// TIA Portal V16 export
// export: Created 2021-09-08T12:46:11.6644631Z, ExportSetting WithDefaults, DisplayName Totally Integrated Automation Portal, DisplayVersion V16 Update 3, DisplayName TIA Portal Version Control Interface, DisplayVersion V16 Update 2, DisplayName TIA Portal Openness, DisplayVersion V16 Update 3, DisplayName TIA Portal Teamcenter Gateway, DisplayVersion V16, DisplayName STEP 7 Professional, DisplayVersion V16 Update 3, DisplayName STEP 7 Safety, DisplayVersion V16, DisplayName WinCC Advanced, DisplayVersion V16 Update 3
FUNCTION_BLOCK "AllPump"   // FB2, FBD
{ S7_Optimized_Access := 'TRUE' }
VERSION : 0.1
// stored: AutoNumber true, IsIECCheckEnabled false, IsRetainMemResEnabled false, MemoryReserve 100, SetENOAutomatically false, UDAEnableTagReadback false
   VAR
      PU30x { S7_SetPoint := 'True'} : "PumpCntrl2Pu1Fc";
      cmUZ_P30x { S7_SetPoint := 'True'} : Bool;
      cmUZ_P120x : Bool;
      cmUZ_P150x : Bool;
      tmrLowPresP30x { S7_SetPoint := 'True'} : TON_TIME;
      tmrLowFreqP30x { S7_SetPoint := 'True'} : TON_TIME;
      tLowPresP30x { S7_SetPoint := 'True'} : Time;
      tLowFreqP30x : Time;
      PU120x { S7_SetPoint := 'True'} : "PumpCntrl2Pu1Fc";
      tmrLowPresP120x { S7_SetPoint := 'True'} : TON_TIME;
      tLowPresP120x { S7_SetPoint := 'True'} : Time;
      tNoPulseP120x : Time;
      PU150x { S7_SetPoint := 'True'} : "PumpCntrl2Pu1Fc";
      tmrLowPresP150x { S7_SetPoint := 'True'} : TON_TIME;
      tLowPresP150x { S7_SetPoint := 'True'} : Time;
      tNoPulseP150x : Time;
      noPulseTOF_P120x { S7_SetPoint := 'True'} : "noPulseTOF";
      noPulseTOF_P150x { S7_SetPoint := 'True'} : "noPulseTOF";
      P701 { S7_SetPoint := 'True'} : "PumpCntr";
      P702 { S7_SetPoint := 'True'} : "PumpCntr";
      P901 { S7_SetPoint := 'True'} : "PumpCntr";
      P1301 { S7_SetPoint := 'True'} : "PumpCntr";
      P2001 { S7_SetPoint := 'True'} : "PumpCntr";
      C501 { S7_SetPoint := 'True'} : "PumpCntr";
      sel2pu_P70x { S7_SetPoint := 'True'} : "sel2pu";
   END_VAR
BEGIN

REGION Network 1: P30x - выбор рабочего
   // Помилка датчиків рівня TW201, TW202
   // Аварійно низький рівень TW201, TW202
   // Помилка датчика PT301
   // Аварійно низьке значення PT301
   // Аварійно високе значення PT301
   // Помилка датчика PT401
   // Аварійно низьке значення PT401
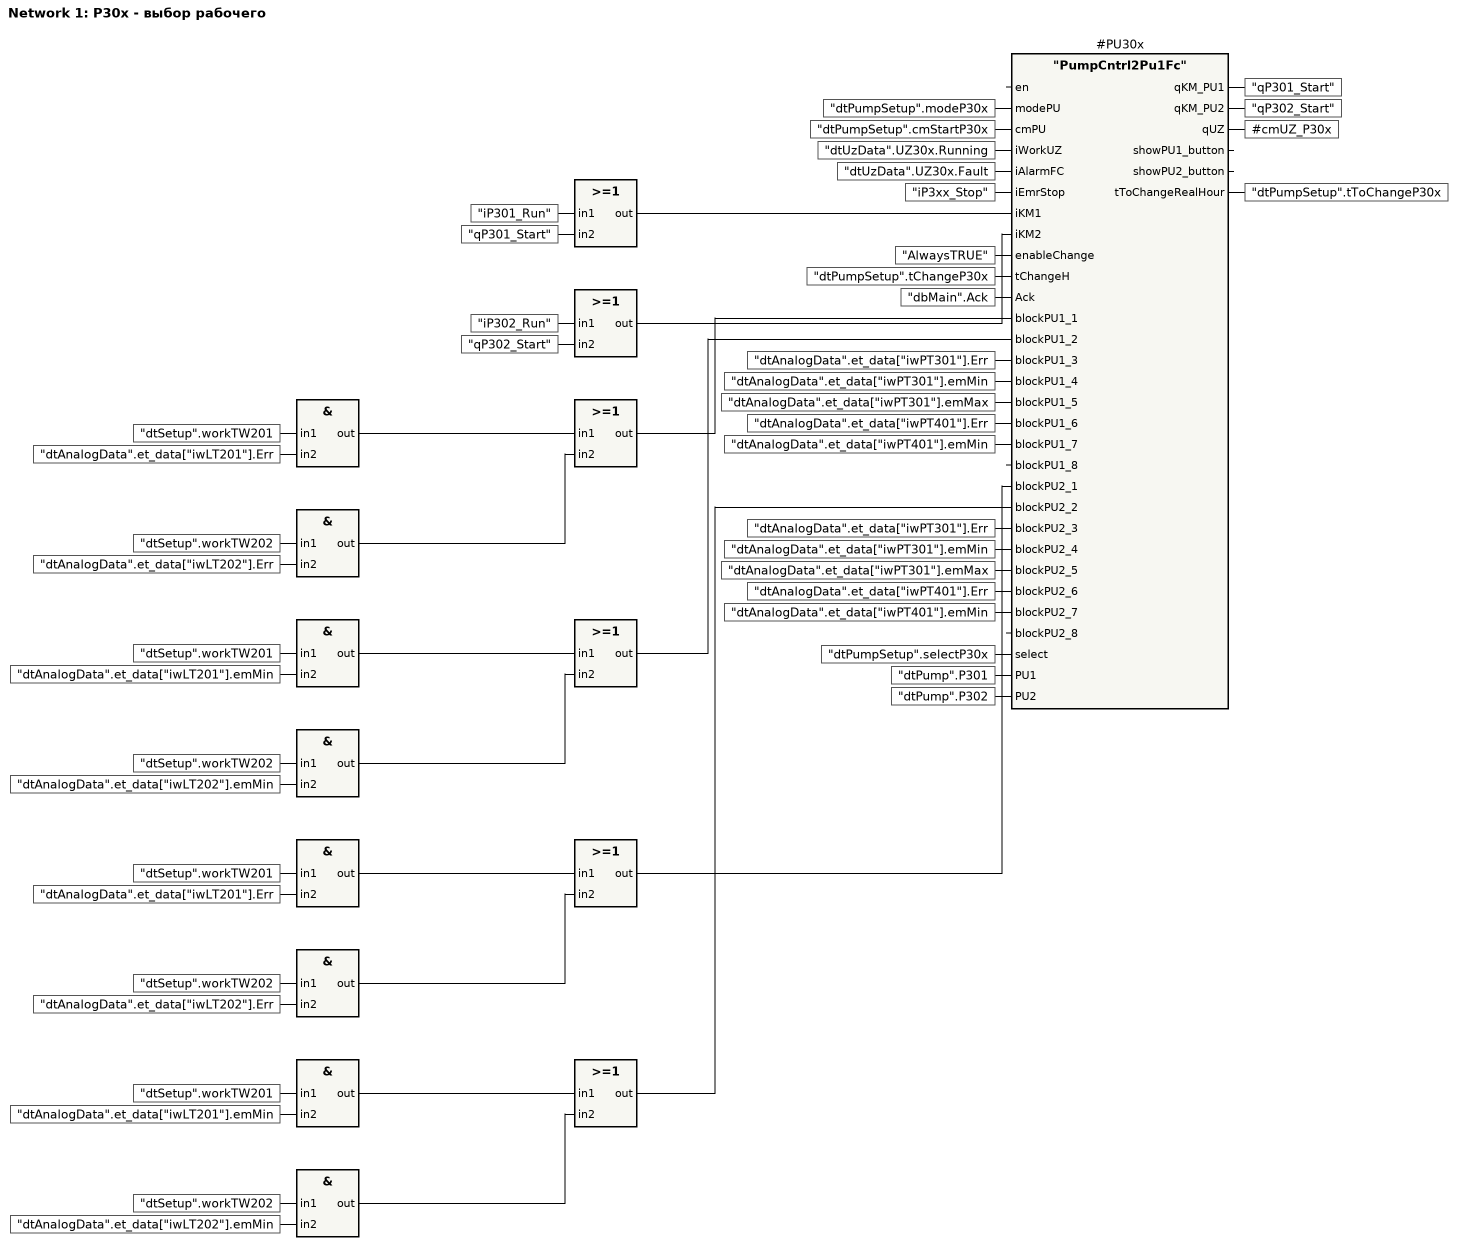
   #PU30x(modePU := "dtPumpSetup".modeP30x,   // "PumpCntrl2Pu1Fc"
          cmPU := "dtPumpSetup".cmStartP30x,
          iWorkUZ := "dtUzData".UZ30x.Running,
          iAlarmFC := "dtUzData".UZ30x.Fault,
          iEmrStop := "iP3xx_Stop",
          iKM1 := "iP301_Run" OR "qP301_Start",
          iKM2 := "iP302_Run" OR "qP302_Start",
          enableChange := "AlwaysTRUE",
          tChangeH := "dtPumpSetup".tChangeP30x,
          Ack := "dbMain".Ack,
          blockPU1_1 := ("dtSetup".workTW201 AND "dtAnalogData".et_data["iwLT201"].Err) OR ("dtSetup".workTW202 AND "dtAnalogData".et_data["iwLT202"].Err),
          blockPU1_2 := ("dtSetup".workTW201 AND "dtAnalogData".et_data["iwLT201"].emMin) OR ("dtSetup".workTW202 AND "dtAnalogData".et_data["iwLT202"].emMin),
          blockPU1_3 := "dtAnalogData".et_data["iwPT301"].Err,
          blockPU1_4 := "dtAnalogData".et_data["iwPT301"].emMin,
          blockPU1_5 := "dtAnalogData".et_data["iwPT301"].emMax,
          blockPU1_6 := "dtAnalogData".et_data["iwPT401"].Err,
          blockPU1_7 := "dtAnalogData".et_data["iwPT401"].emMin,
          blockPU2_1 := ("dtSetup".workTW201 AND "dtAnalogData".et_data["iwLT201"].Err) OR ("dtSetup".workTW202 AND "dtAnalogData".et_data["iwLT202"].Err),
          blockPU2_2 := ("dtSetup".workTW201 AND "dtAnalogData".et_data["iwLT201"].emMin) OR ("dtSetup".workTW202 AND "dtAnalogData".et_data["iwLT202"].emMin),
          blockPU2_3 := "dtAnalogData".et_data["iwPT301"].Err,
          blockPU2_4 := "dtAnalogData".et_data["iwPT301"].emMin,
          blockPU2_5 := "dtAnalogData".et_data["iwPT301"].emMax,
          blockPU2_6 := "dtAnalogData".et_data["iwPT401"].Err,
          blockPU2_7 := "dtAnalogData".et_data["iwPT401"].emMin,
          select := "dtPumpSetup".selectP30x,
          PU1 := "dtPump".P301,
          PU2 := "dtPump".P302,
          qKM_PU1 => "qP301_Start",
          qKM_PU2 => "qP302_Start",
          qUZ => #cmUZ_P30x,
          tToChangeRealHour => "dtPumpSetup".tToChangeP30x);
END_REGION

REGION Network 2: P30x - частотник
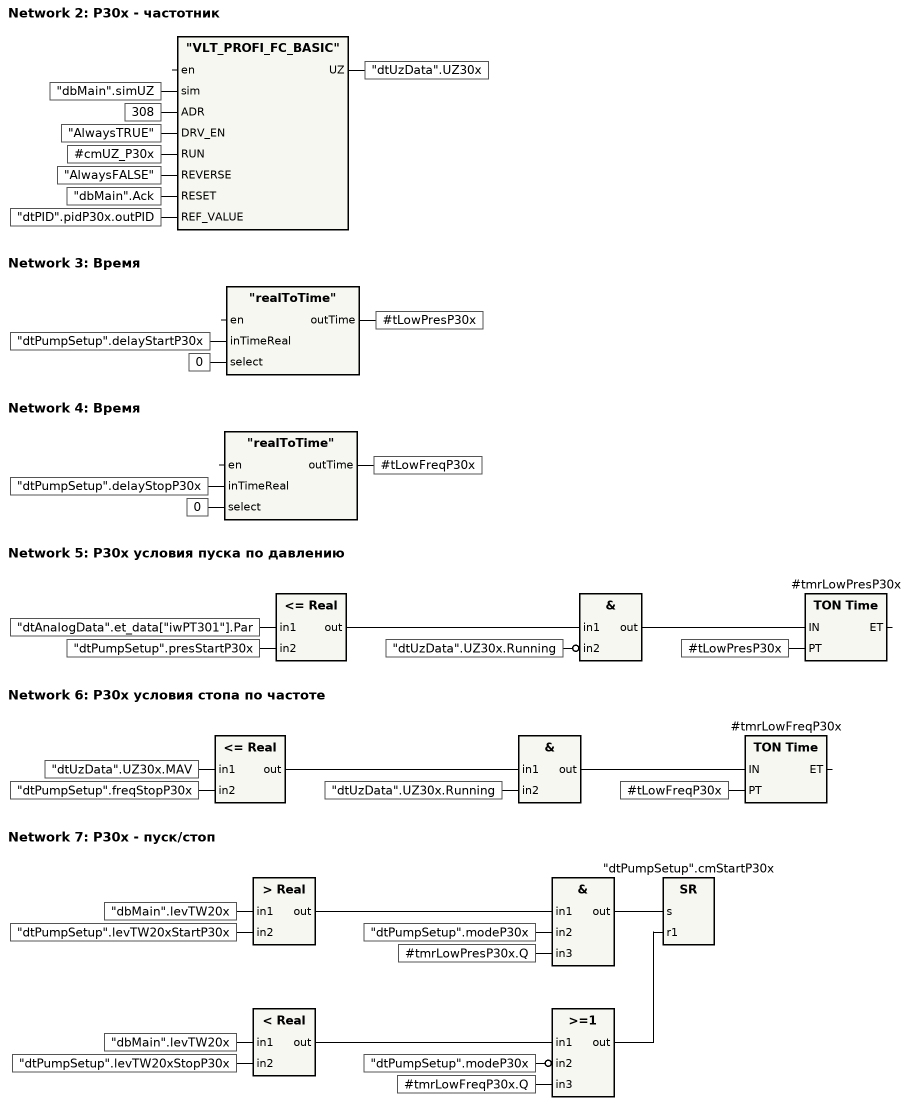
   "VLT_PROFI_FC_BASIC"(sim := "dbMain".simUZ,
                        ADR := 308,
                        DRV_EN := "AlwaysTRUE",
                        RUN := #cmUZ_P30x,
                        REVERSE := "AlwaysFALSE",
                        RESET := "dbMain".Ack,
                        REF_VALUE := "dtPID".pidP30x.outPID,
                        UZ => "dtUzData".UZ30x);
END_REGION

REGION Network 3: Время
   "realToTime"(inTimeReal := "dtPumpSetup".delayStartP30x, select := 0, outTime => #tLowPresP30x);
END_REGION

REGION Network 4: Время
   "realToTime"(inTimeReal := "dtPumpSetup".delayStopP30x, select := 0, outTime => #tLowFreqP30x);
END_REGION

REGION Network 5: P30x условия пуска по давлению
   #tmrLowPresP30x(IN := ("dtAnalogData".et_data["iwPT301"].Par <= "dtPumpSetup".presStartP30x) AND NOT "dtUzData".UZ30x.Running,   // TON
                   PT := #tLowPresP30x);
END_REGION

REGION Network 6: P30x условия стопа по частоте
   #tmrLowFreqP30x(IN := ("dtUzData".UZ30x.MAV <= "dtPumpSetup".freqStopP30x) AND "dtUzData".UZ30x.Running,   // TON
                   PT := #tLowFreqP30x);
END_REGION

REGION Network 7: P30x - пуск/стоп
   IF ("dbMain".levTW20x > "dtPumpSetup".levTW20xStartP30x) AND "dtPumpSetup".modeP30x AND #tmrLowPresP30x.Q THEN
       "dtPumpSetup".cmStartP30x := TRUE;   // SR flip-flop
   END_IF;
   IF ("dbMain".levTW20x < "dtPumpSetup".levTW20xStopP30x) OR NOT "dtPumpSetup".modeP30x OR #tmrLowFreqP30x.Q THEN
       "dtPumpSetup".cmStartP30x := FALSE;
   END_IF;
END_REGION

REGION Network 8: -------------------------------------------------P1201, 1202
END_REGION

REGION Network 9: P120x - выбор рабочего !!!!!!!!!!!!!!!!!!!!!!!!!!!!!!!!!!!!!!!!!!!!!!!!!! Убрать iP1201_run
   // Помилка датчиків рівня LT1101
   // Аварійно низький рівень TW1101
   // Помилка датчика PT1201
   // Аварійно низьке значення PT1201
   // Аварійно високе значення PT1201
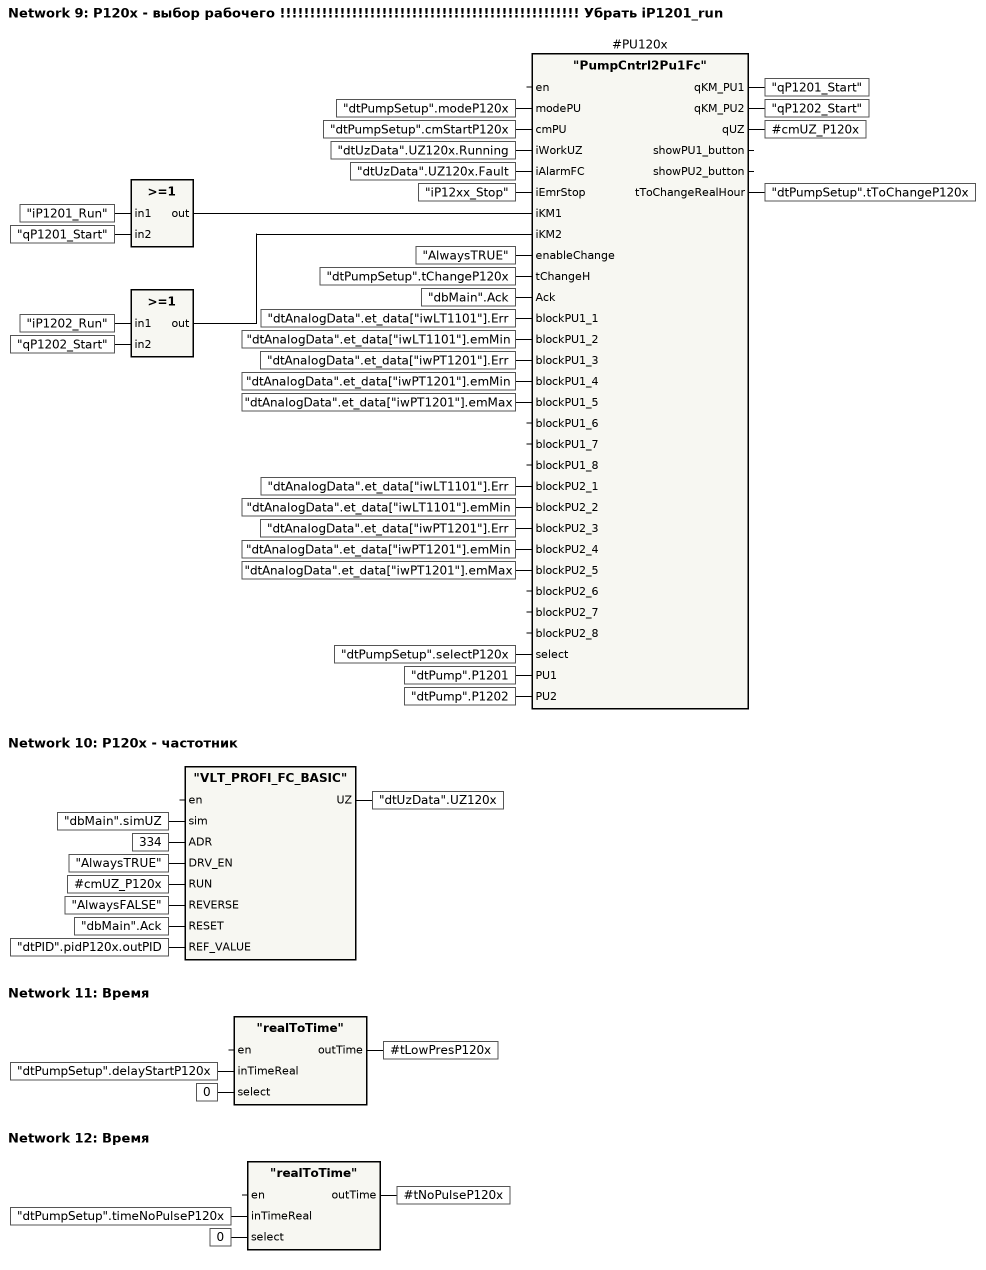
   #PU120x(modePU := "dtPumpSetup".modeP120x,   // "PumpCntrl2Pu1Fc"
           cmPU := "dtPumpSetup".cmStartP120x,
           iWorkUZ := "dtUzData".UZ120x.Running,
           iAlarmFC := "dtUzData".UZ120x.Fault,
           iEmrStop := "iP12xx_Stop",
           iKM1 := "iP1201_Run" OR "qP1201_Start",
           iKM2 := "iP1202_Run" OR "qP1202_Start",
           enableChange := "AlwaysTRUE",
           tChangeH := "dtPumpSetup".tChangeP120x,
           Ack := "dbMain".Ack,
           blockPU1_1 := "dtAnalogData".et_data["iwLT1101"].Err,
           blockPU1_2 := "dtAnalogData".et_data["iwLT1101"].emMin,
           blockPU1_3 := "dtAnalogData".et_data["iwPT1201"].Err,
           blockPU1_4 := "dtAnalogData".et_data["iwPT1201"].emMin,
           blockPU1_5 := "dtAnalogData".et_data["iwPT1201"].emMax,
           blockPU2_1 := "dtAnalogData".et_data["iwLT1101"].Err,
           blockPU2_2 := "dtAnalogData".et_data["iwLT1101"].emMin,
           blockPU2_3 := "dtAnalogData".et_data["iwPT1201"].Err,
           blockPU2_4 := "dtAnalogData".et_data["iwPT1201"].emMin,
           blockPU2_5 := "dtAnalogData".et_data["iwPT1201"].emMax,
           select := "dtPumpSetup".selectP120x,
           PU1 := "dtPump".P1201,
           PU2 := "dtPump".P1202,
           qKM_PU1 => "qP1201_Start",
           qKM_PU2 => "qP1202_Start",
           qUZ => #cmUZ_P120x,
           tToChangeRealHour => "dtPumpSetup".tToChangeP120x);
END_REGION

REGION Network 10: P120x - частотник
   "VLT_PROFI_FC_BASIC"(sim := "dbMain".simUZ,
                        ADR := 334,
                        DRV_EN := "AlwaysTRUE",
                        RUN := #cmUZ_P120x,
                        REVERSE := "AlwaysFALSE",
                        RESET := "dbMain".Ack,
                        REF_VALUE := "dtPID".pidP120x.outPID,
                        UZ => "dtUzData".UZ120x);
END_REGION

REGION Network 11: Время
   "realToTime"(inTimeReal := "dtPumpSetup".delayStartP120x, select := 0, outTime => #tLowPresP120x);
END_REGION

REGION Network 12: Время
   "realToTime"(inTimeReal := "dtPumpSetup".timeNoPulseP120x, select := 0, outTime => #tNoPulseP120x);
END_REGION

REGION Network 13: P120x условия пуска по давлению
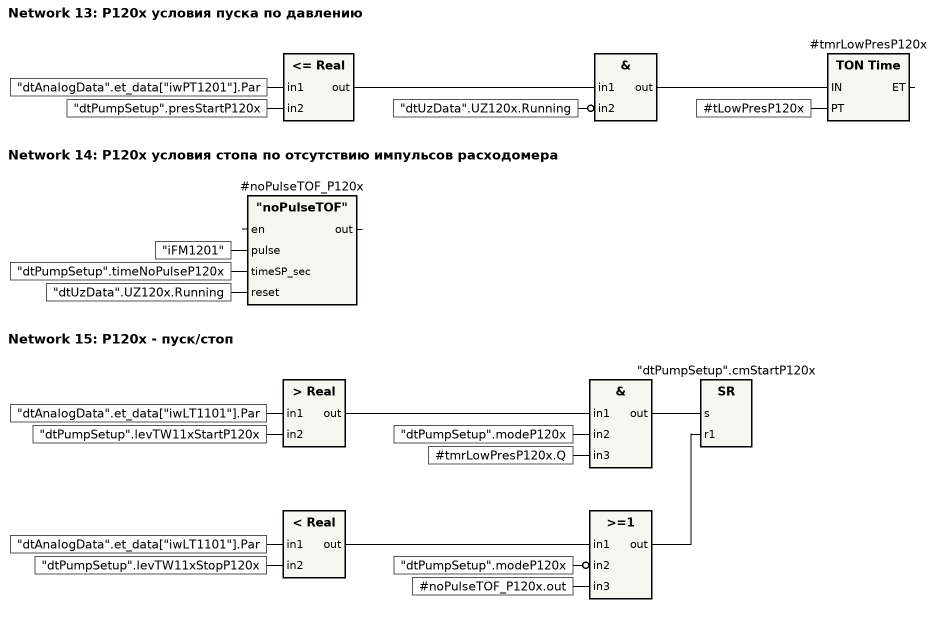
   #tmrLowPresP120x(IN := ("dtAnalogData".et_data["iwPT1201"].Par <= "dtPumpSetup".presStartP120x) AND NOT "dtUzData".UZ120x.Running,   // TON
                    PT := #tLowPresP120x);
END_REGION

REGION Network 14: P120x условия стопа по отсутствию импульсов расходомера
   #noPulseTOF_P120x(pulse := "iFM1201",   // "noPulseTOF"
                     timeSP_sec := "dtPumpSetup".timeNoPulseP120x,
                     reset := "dtUzData".UZ120x.Running);
END_REGION

REGION Network 15: P120x - пуск/стоп
   IF ("dtAnalogData".et_data["iwLT1101"].Par > "dtPumpSetup".levTW11xStartP120x) AND "dtPumpSetup".modeP120x AND #tmrLowPresP120x.Q THEN
       "dtPumpSetup".cmStartP120x := TRUE;   // SR flip-flop
   END_IF;
   IF ("dtAnalogData".et_data["iwLT1101"].Par < "dtPumpSetup".levTW11xStopP120x) OR NOT "dtPumpSetup".modeP120x OR #noPulseTOF_P120x.out THEN
       "dtPumpSetup".cmStartP120x := FALSE;
   END_IF;
END_REGION

REGION Network 16: -------------------------------------------------P1501, 1502
END_REGION

REGION Network 17: P150x - выбор рабочего !!!!!!!!!!!!!!!!!!!!!!!!!!!!!!!!!!!!!!!!!!!!!!!!!! Убрать iP1501_run
   // Помилка датчиків рівня TW1401, TW1402
   // Аварійно низький рівень TW1401, TW1402
   // Помилка датчика PT1501
   // Аварійно низьке значення PT1501
   // Аварійно високе значення PT1501
   // Помилка датчика PT1701
   // Аварійно низьке значення PT1701
   // Аварійно високе значення PT1701
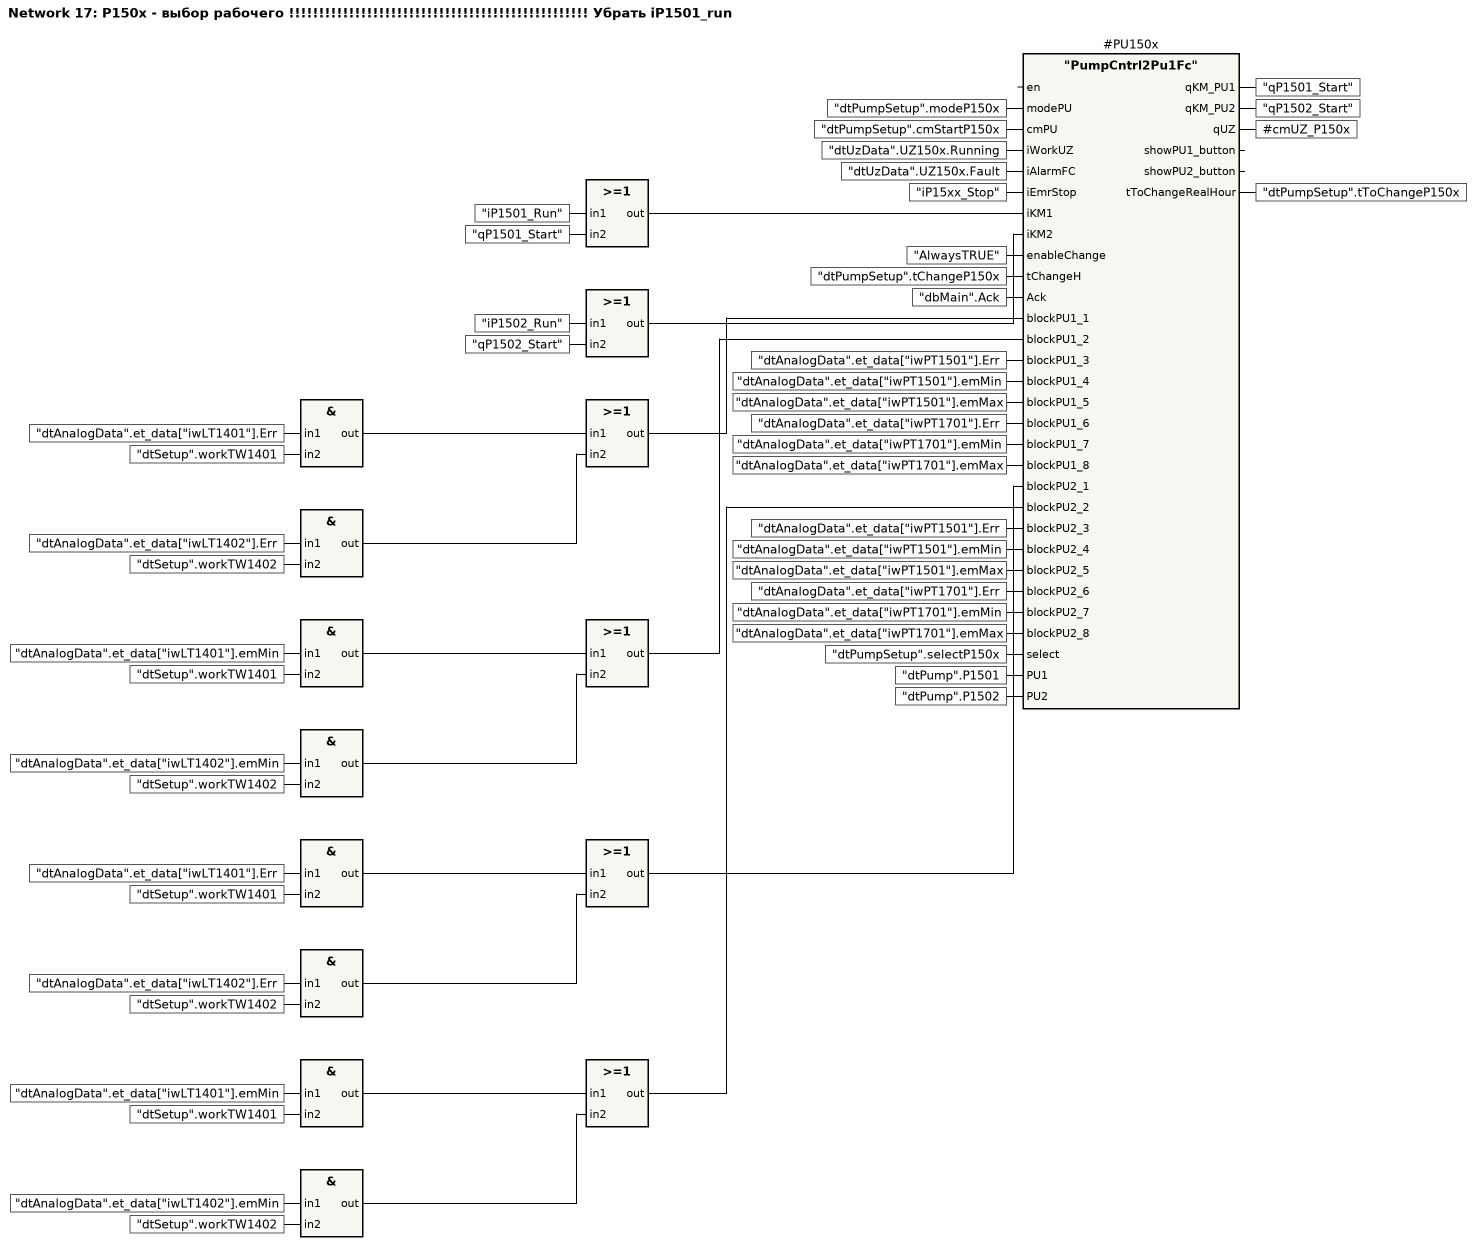
   #PU150x(modePU := "dtPumpSetup".modeP150x,   // "PumpCntrl2Pu1Fc"
           cmPU := "dtPumpSetup".cmStartP150x,
           iWorkUZ := "dtUzData".UZ150x.Running,
           iAlarmFC := "dtUzData".UZ150x.Fault,
           iEmrStop := "iP15xx_Stop",
           iKM1 := "iP1501_Run" OR "qP1501_Start",
           iKM2 := "iP1502_Run" OR "qP1502_Start",
           enableChange := "AlwaysTRUE",
           tChangeH := "dtPumpSetup".tChangeP150x,
           Ack := "dbMain".Ack,
           blockPU1_1 := ("dtAnalogData".et_data["iwLT1401"].Err AND "dtSetup".workTW1401) OR ("dtAnalogData".et_data["iwLT1402"].Err AND "dtSetup".workTW1402),
           blockPU1_2 := ("dtAnalogData".et_data["iwLT1401"].emMin AND "dtSetup".workTW1401) OR ("dtAnalogData".et_data["iwLT1402"].emMin AND "dtSetup".workTW1402),
           blockPU1_3 := "dtAnalogData".et_data["iwPT1501"].Err,
           blockPU1_4 := "dtAnalogData".et_data["iwPT1501"].emMin,
           blockPU1_5 := "dtAnalogData".et_data["iwPT1501"].emMax,
           blockPU1_6 := "dtAnalogData".et_data["iwPT1701"].Err,
           blockPU1_7 := "dtAnalogData".et_data["iwPT1701"].emMin,
           blockPU1_8 := "dtAnalogData".et_data["iwPT1701"].emMax,
           blockPU2_1 := ("dtAnalogData".et_data["iwLT1401"].Err AND "dtSetup".workTW1401) OR ("dtAnalogData".et_data["iwLT1402"].Err AND "dtSetup".workTW1402),
           blockPU2_2 := ("dtAnalogData".et_data["iwLT1401"].emMin AND "dtSetup".workTW1401) OR ("dtAnalogData".et_data["iwLT1402"].emMin AND "dtSetup".workTW1402),
           blockPU2_3 := "dtAnalogData".et_data["iwPT1501"].Err,
           blockPU2_4 := "dtAnalogData".et_data["iwPT1501"].emMin,
           blockPU2_5 := "dtAnalogData".et_data["iwPT1501"].emMax,
           blockPU2_6 := "dtAnalogData".et_data["iwPT1701"].Err,
           blockPU2_7 := "dtAnalogData".et_data["iwPT1701"].emMin,
           blockPU2_8 := "dtAnalogData".et_data["iwPT1701"].emMax,
           select := "dtPumpSetup".selectP150x,
           PU1 := "dtPump".P1501,
           PU2 := "dtPump".P1502,
           qKM_PU1 => "qP1501_Start",
           qKM_PU2 => "qP1502_Start",
           qUZ => #cmUZ_P150x,
           tToChangeRealHour => "dtPumpSetup".tToChangeP150x);
END_REGION

REGION Network 18: P150x - частотник
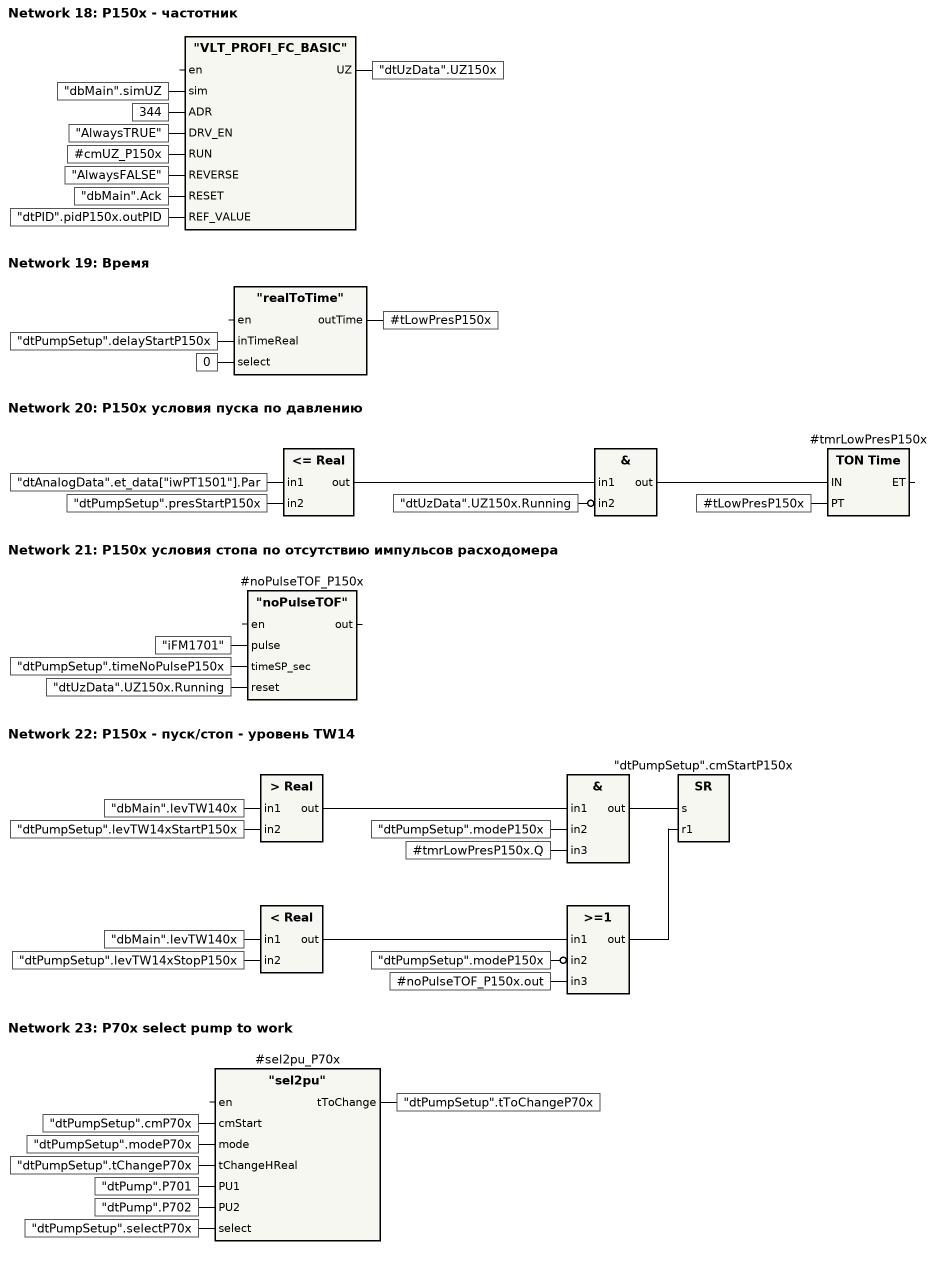
   "VLT_PROFI_FC_BASIC"(sim := "dbMain".simUZ,
                        ADR := 344,
                        DRV_EN := "AlwaysTRUE",
                        RUN := #cmUZ_P150x,
                        REVERSE := "AlwaysFALSE",
                        RESET := "dbMain".Ack,
                        REF_VALUE := "dtPID".pidP150x.outPID,
                        UZ => "dtUzData".UZ150x);
END_REGION

REGION Network 19: Время
   "realToTime"(inTimeReal := "dtPumpSetup".delayStartP150x, select := 0, outTime => #tLowPresP150x);
END_REGION

REGION Network 20: P150x условия пуска по давлению
   #tmrLowPresP150x(IN := ("dtAnalogData".et_data["iwPT1501"].Par <= "dtPumpSetup".presStartP150x) AND NOT "dtUzData".UZ150x.Running,   // TON
                    PT := #tLowPresP150x);
END_REGION

REGION Network 21: P150x условия стопа по отсутствию импульсов расходомера
   #noPulseTOF_P150x(pulse := "iFM1701",   // "noPulseTOF"
                     timeSP_sec := "dtPumpSetup".timeNoPulseP150x,
                     reset := "dtUzData".UZ150x.Running);
END_REGION

REGION Network 22: P150x - пуск/стоп - уровень TW14
   IF ("dbMain".levTW140x > "dtPumpSetup".levTW14xStartP150x) AND "dtPumpSetup".modeP150x AND #tmrLowPresP150x.Q THEN
       "dtPumpSetup".cmStartP150x := TRUE;   // SR flip-flop
   END_IF;
   IF ("dbMain".levTW140x < "dtPumpSetup".levTW14xStopP150x) OR NOT "dtPumpSetup".modeP150x OR #noPulseTOF_P150x.out THEN
       "dtPumpSetup".cmStartP150x := FALSE;
   END_IF;
END_REGION

REGION Network 23: P70x select pump to work
   #sel2pu_P70x(cmStart := "dtPumpSetup".cmP70x,   // "sel2pu"
                mode := "dtPumpSetup".modeP70x,
                tChangeHReal := "dtPumpSetup".tChangeP70x,
                PU1 := "dtPump".P701,
                PU2 := "dtPump".P702,
                select := "dtPumpSetup".selectP70x,
                tToChange => "dtPumpSetup".tToChangeP70x);
END_REGION

REGION Network 24: P701
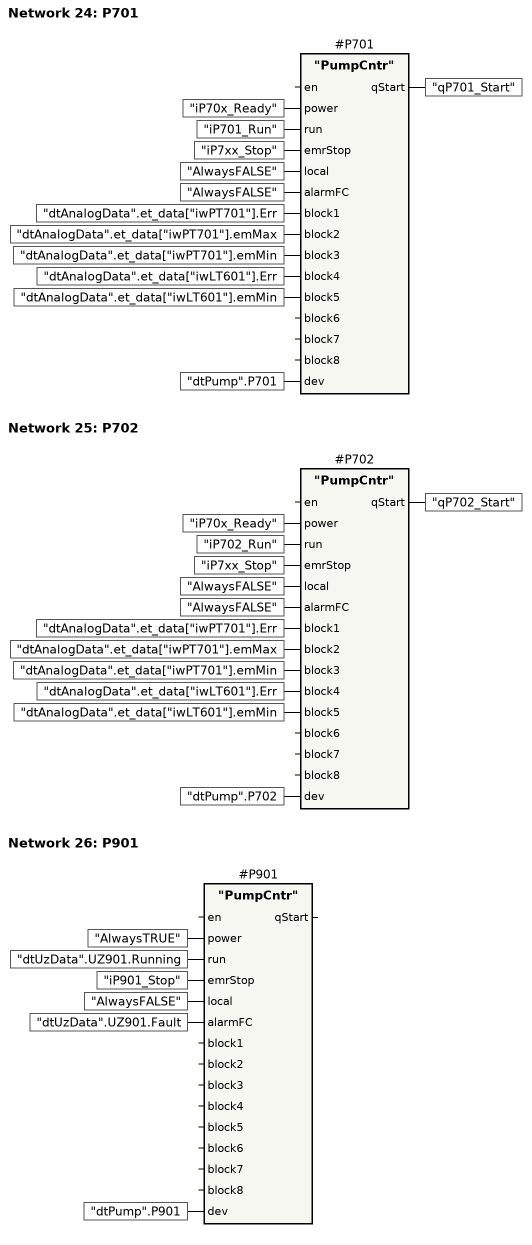
   #P701(power := "iP70x_Ready",   // "PumpCntr"
         run := "iP701_Run",
         emrStop := "iP7xx_Stop",
         local := "AlwaysFALSE",
         alarmFC := "AlwaysFALSE",
         block1 := "dtAnalogData".et_data["iwPT701"].Err,
         block2 := "dtAnalogData".et_data["iwPT701"].emMax,
         block3 := "dtAnalogData".et_data["iwPT701"].emMin,
         block4 := "dtAnalogData".et_data["iwLT601"].Err,
         block5 := "dtAnalogData".et_data["iwLT601"].emMin,
         dev := "dtPump".P701,
         qStart => "qP701_Start");
END_REGION

REGION Network 25: P702
   #P702(power := "iP70x_Ready",   // "PumpCntr"
         run := "iP702_Run",
         emrStop := "iP7xx_Stop",
         local := "AlwaysFALSE",
         alarmFC := "AlwaysFALSE",
         block1 := "dtAnalogData".et_data["iwPT701"].Err,
         block2 := "dtAnalogData".et_data["iwPT701"].emMax,
         block3 := "dtAnalogData".et_data["iwPT701"].emMin,
         block4 := "dtAnalogData".et_data["iwLT601"].Err,
         block5 := "dtAnalogData".et_data["iwLT601"].emMin,
         dev := "dtPump".P702,
         qStart => "qP702_Start");
END_REGION

REGION Network 26: P901
   #P901(power := "AlwaysTRUE",   // "PumpCntr"
         run := "dtUzData".UZ901.Running,
         emrStop := "iP901_Stop",
         local := "AlwaysFALSE",
         alarmFC := "dtUzData".UZ901.Fault,
         dev := "dtPump".P901);
END_REGION

REGION Network 27: P901 - частотник
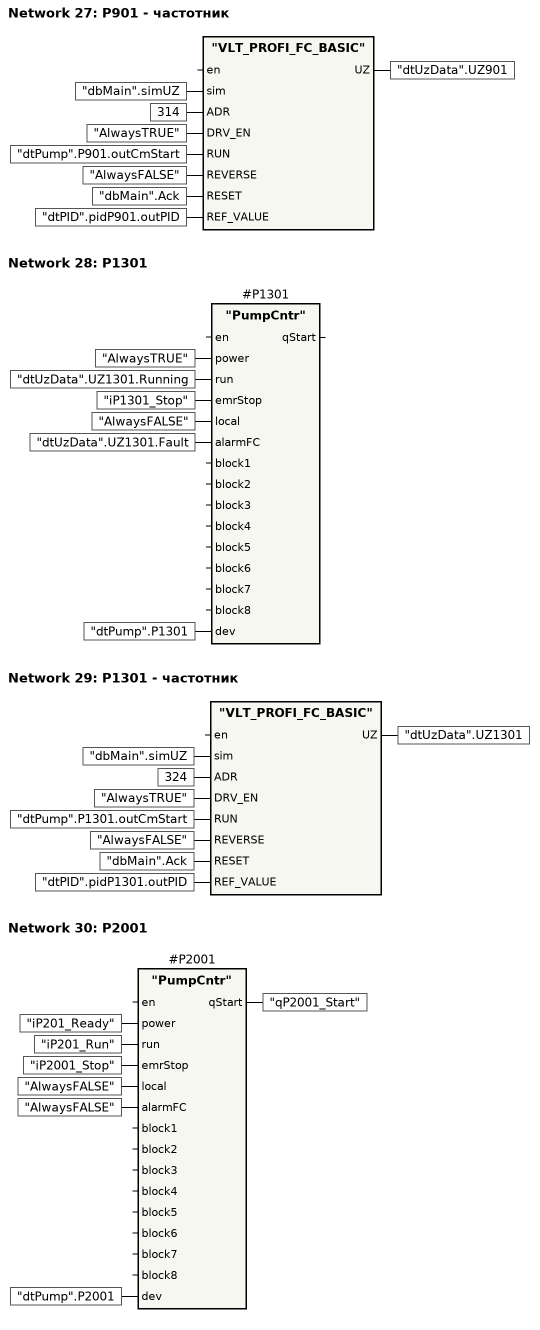
   "VLT_PROFI_FC_BASIC"(sim := "dbMain".simUZ,
                        ADR := 314,
                        DRV_EN := "AlwaysTRUE",
                        RUN := "dtPump".P901.outCmStart,
                        REVERSE := "AlwaysFALSE",
                        RESET := "dbMain".Ack,
                        REF_VALUE := "dtPID".pidP901.outPID,
                        UZ => "dtUzData".UZ901);
END_REGION

REGION Network 28: P1301
   #P1301(power := "AlwaysTRUE",   // "PumpCntr"
          run := "dtUzData".UZ1301.Running,
          emrStop := "iP1301_Stop",
          local := "AlwaysFALSE",
          alarmFC := "dtUzData".UZ1301.Fault,
          dev := "dtPump".P1301);
END_REGION

REGION Network 29: P1301 - частотник
   "VLT_PROFI_FC_BASIC"(sim := "dbMain".simUZ,
                        ADR := 324,
                        DRV_EN := "AlwaysTRUE",
                        RUN := "dtPump".P1301.outCmStart,
                        REVERSE := "AlwaysFALSE",
                        RESET := "dbMain".Ack,
                        REF_VALUE := "dtPID".pidP1301.outPID,
                        UZ => "dtUzData".UZ1301);
END_REGION

REGION Network 30: P2001
   #P2001(power := "iP201_Ready",   // "PumpCntr"
          run := "iP201_Run",
          emrStop := "iP2001_Stop",
          local := "AlwaysFALSE",
          alarmFC := "AlwaysFALSE",
          dev := "dtPump".P2001,
          qStart => "qP2001_Start");
END_REGION
END_FUNCTION_BLOCK
